PROGRAM PRG_FlyingSaw
VAR
	nState: INT;

	sMsg: STRING(INT#30);
END_VAR

rProcessActive(CLK:= bProcessActive , Q=> );
IF rProcessActive.Q THEN
			i	:= i+1;
END_IF

CASE nState OF
	
0:
	IF bStartSensor THEN
		nState	:= 5;
		bProcessActive	:= TRUE;
	END_IF

5:
	IF stAxis1.OUT.bEnabled AND stAxis2.OUT.bEnabled AND stAxis3.OUT.bEnabled THEN
		nState	:= 10;	
	END_IF
	
10:	
	stAxis1.IN.bMoveAbs		:= TRUE;
	stAxis1.IN.fVelo				:= 3000;
	stAxis1.IN.fPos					:= 20000;
	IF stAxis1.OUT.bMoveAbsBusy AND NOT stAxis1.OUT.bMoveAbsErr THEN
		nState						:= 20;
		//stAxis1.IN.bMcMoveModulo	:= FALSE;
	ELSIF stAxis1.OUT.bMoveAbsErr THEN
		nLastState					:= nState;		
		stAxis1.IN.bMcMoveModulo	:= FALSE;
		nState						:= 999;
	END_IF
	
20:
	fCalculate	:= (((DINT_TO_LREAL(i-1))*20000)+1000);
	IF Axis1.NcToPlc.ModuloActPos >= 1000 THEN
		nState	:= 30;
	ELSIF axis1.Status.Error THEN
		nState	:= 999;
	END_IF
	
30:
	stAxis1.IN.bGearInPos			:= TRUE;
	stAxis1.IN.fMasterGearPos		:= 6000;
	stAxis1.IN.fSlaveGearPos		:= 1000;

	(*
	IF i=1 THEN
		stAxis1.IN.fMasterGearPos		:= 6000;
		stAxis1.IN.fSlaveGearPos		:= 1000;
		stAxis1.IN.fMasterStartDistance	:= 0;
	ELSE
		stAxis1.IN.fMasterGearPos		:= 6000+(20000*DINT_TO_LREAL(i));
		stAxis1.IN.fSlaveGearPos		:= 1000;
		stAxis1.IN.fMasterStartDistance	:= 20000*i;
	END_IF*)
	IF stAxis1.OUT.bCoupled AND NOT stAxis1.OUT.bCoupleErr THEN
		nState					:= 40;
		stAxis1.IN.bGearInPos	:= FALSE;
		sMsg					:= 'Flying Saw Hareketi Basladi...';
	ELSIF stAxis1.OUT.bCoupleErr THEN
	//	stAxis1.IN.bGearInPos	:= FALSE;
		nState					:= 999;
	END_IF
	
40:	
	IF Axis2.NcToPlc.ActPos>=1000 THEN
		nState		:= 50;
	ELSIF axis2.Status.Error THEN
		nState		:= 999;
	END_IF
		
50:
	stAxis3.IN.bMoveAbs				:= TRUE;
	stAxis3.IN.fVelo				:= 2000;
	stAxis3.IN.fPos					:= 1000;
	IF stAxis3.OUT.bMoveAbsBusy AND NOT stAxis3.OUT.bMoveAbsErr THEN
		nState				:= 60;
		stAxis3.IN.bMoveAbs	:= FALSE;
	ELSIF stAxis3.OUT.bMoveAbsErr THEN
		nState				:= 999;
		stAxis3.IN.bMoveAbs	:= FALSE;
	END_IF

60:
	IF stAxis3.OUT.bMoveAbsDone  AND NOT stAxis3.OUT.bMoveAbsErr  THEN
		nState				:= 70;
	ELSIF stAxis3.OUT.bMoveAbsErr  THEN
		nState				:= 999;
	END_IF
	
70:
	stAxis3.IN.bMoveAbs		:= TRUE;
	stAxis3.IN.fVelo		:= 1000;
	stAxis3.IN.fPos			:= 0;
	IF stAxis3.OUT.bMoveAbsBusy AND NOT stAxis3.OUT.bMoveAbsErr THEN
		nState				:= 80;
		stAxis3.IN.bMoveAbs	:= FALSE;
	ELSIF stAxis3.OUT.bMoveAbsErr THEN
		nState				:= 999;
		stAxis3.IN.bMoveAbs	:= FALSE;
	END_IF
	
80:
	IF stAxis3.OUT.bMoveAbsDone  AND NOT stAxis3.OUT.bMoveAbsErr  THEN
		nState				:= 90;
	ELSIF stAxis3.OUT.bMoveAbsErr  THEN
		nState				:= 999;
	END_IF
	
90:
	stAxis1.IN.bGearOut := TRUE;
	IF stAxis1.OUT.bDecoupled THEN
		stAxis1.IN.bGearOut := FALSE;
		nState				:= 100;
		sMsg				:= 'Flying Saw Hareketi Sonlandi...';
	END_IF
	
100:
	stAxis2.IN.bStop	:= TRUE;
	IF stAxis2.OUT.bStopDone THEN
		nState			:= 110;
		stAxis2.IN.bStop:= FALSE;
	END_IF
	
110:
	stAxis2.IN.bMoveAbs	:= TRUE;
	stAxis2.IN.fVelo	:= 7000;
	stAxis2.IN.fPos		:= 0;
	IF stAxis2.OUT.bMoveAbsBusy AND NOT stAxis2.OUT.bMoveAbsErr  THEN
		nState	:= 120;
	//	stAxis2.IN.bMoveAbs	:= FALSE;	
	ELSIF stAxis2.OUT.bMoveAbsErr  THEN
		nState	:= 99;		
		stAxis2.IN.bMoveAbs	:= FALSE;	
	END_IF
	
120:
	IF stAxis2.OUT.bMoveAbsDone AND NOT stAxis2.OUT.bMoveAbsErr  THEN
		nState	:= 130;
	ELSIF stAxis2.OUT.bMoveAbsErr  THEN
		nState		:= 99;
	END_IF
	

(*	
140:
	stAxis1.IN.bMcMoveModulo		:= TRUE;
	stAxis1.IN.fVelo				:= 2000;
	stAxis1.IN.fPos					:= 0;
	IF stAxis1.OUT.bMoveModuloBusy AND NOT stAxis1.OUT.bMoveModuloErr THEN
		nState						:= 150;
		stAxis1.IN.bMcMoveModulo	:= FALSE;
	ELSIF stAxis1.OUT.bMoveModuloErr THEN
		nLastState					:= nState;		
		stAxis1.IN.bMcMoveModulo	:= FALSE;
		nState						:= 999;
	END_IF
	
150:
	IF stAxis1.OUT.bMoveModuloDone THEN
		nState			:= 160;
		bProcessActive	:= FALSE;
	ELSIF stAxis1.OUT.bMoveModuloErr THEN
		nState			:= 999;
	END_IF
	*)
160:
	stAxis1.IN.bSetPosition		:= TRUE;
	IF stAxis1.OUT.bSetPositionDone THEN
		stAxis1.IN.bSetPosition	:= FALSE;
		nState					:= 0;
		bProcessActive			:= FALSE;
	END_IF
	
999:
;

END_CASE

IF stAxis1.OUT.bMoveAbsDone AND stAxis2.OUT.bMoveAbsDone  THEN
	nState	:= 160;
	stAxis1.IN.bMoveAbs	:= FALSE;		
	stAxis2.IN.bMoveAbs	:= FALSE;	
ELSIF stAxis1.OUT.bMoveAbsErr THEN
	nState	:= 999;
	stAxis1.IN.bMoveAbs	:= FALSE;	
END_IF


IF NOT bProcessActive AND NOT bStartSensor AND bMalzemeSensoru THEN
		bAsagi		:= TRUE;
		bYukari		:= FALSE;
ELSIF bStartSensor THEN
		bAsagi		:= FALSE;
		bYukari		:= TRUE;
ELSIF bYukariSensor THEN
		bYukari		:= FALSE;
		bAsagi		:= FALSE;
END_IF

END_PROGRAM

(* stored: Version 1.1.0.1, ProductVersion 3.1.4022.12
   POU PRG_FlyingSaw: Id {db73d7f3-ac42-401a-8734-5a44ca8e46a7}, SpecialFunc None *)
